// TIA Portal V19 export
DATA_BLOCK "A02_HMI_IDB"   // DB189
AUTHOR : Piemme
FAMILY : System
// stored: InstanceOfName A02_HMI_FB, InstanceOfType FB
"A02_HMI_FB"
   // VAR
   //    MB2_Decoder { ExternalAccessible := 'False'; ExternalVisible := 'False'; ExternalWritable := 'False'} : "ButtonsHMIDecoder";
   // END_VAR
BEGIN
END_DATA_BLOCK
